// Mitsubishi GX Works2 project: pcl_6   PLC: FX3G

// global labels: Global1
VAR_GLOBAL
  start_day AT X010 : BOOL;
  finish_bread AT M1 : BOOL;
  finish_hala AT M1 : BOOL;
  flour_start_day AT D1100 : REAL;
END_VAR
VAR_GLOBAL CONSTANT
  min_flour : REAL := 100;
END_VAR
VAR_GLOBAL
  is_flour_enough AT M2 : BOOL;
  yeast AT D1200 : REAL;
  flour AT D1100 : REAL;
END_VAR
VAR_GLOBAL CONSTANT
  precent_at_least_5 : REAL := 5;
  precent_at_least_1hlcey5 : REAL := 5;
  precent_at_least_1hlcey2 : REAL := 2;
END_VAR
VAR_GLOBAL
  water AT D1300 : REAL;
END_VAR
VAR_GLOBAL CONSTANT
  hlcey5 : REAL := 5;
  hlcey2 : REAL := 2;
  caul0_3 : REAL := 0.3;
END_VAR
VAR_GLOBAL
  oil AT D1400 : REAL;
END_VAR
VAR_GLOBAL CONSTANT
  caful0_3 : REAL := 0.3;
END_VAR
VAR_GLOBAL
  spises AT D1500 : REAL;
END_VAR
VAR_GLOBAL CONSTANT
  caful0_1 : REAL := 0.1;
END_VAR
VAR_GLOBAL
  is_ingredients_enough AT M3 : BOOL;
  is_water_enough AT M3 : BOOL;
  is_oil_enough AT M4 : BOOL;
  is_spices_enough AT M5 : BOOL;
  spices AT D1500 : REAL;
  is_yeast_enough AT M6 : BOOL;
  day_work AT Y010 : BOOL;
  emergency_button AT M7 : BOOL;
  emergency_button_press AT X007 : BOOL;
  BAKAR AT M9 : BOOL;
  tc1 AT TC200 : BOOL;
END_VAR
VAR_GLOBAL CONSTANT
  cons50 : INT;
  cons500 : REAL := 500;
END_VAR
VAR_GLOBAL
  ts1 AT TS200 : BOOL;
  tc AT TC201 : BOOL;
  tc2 AT TC201 : BOOL;
  ts2 AT TS201 : BOOL;
END_VAR
VAR_GLOBAL CONSTANT
  COUNTER4 : INT;
END_VAR
VAR_GLOBAL
  firctC1 AT CC1 : BOOL;
  outC AT CS1 : BOOL;
  insert_flour AT D1102 : REAL;
  insert_yeast AT D1202 : REAL;
  insert_water AT D1302 : REAL;
  insert_oil AT D1402 : REAL;
  insert_spices AT D1502 : REAL;
  PREPARING AT X002 : BOOL;
  TimerPrep AT TC6 : BOOL;
END_VAR
VAR_GLOBAL CONSTANT
  PT3000 : REAL := 3000;
END_VAR
VAR_GLOBAL
  Lamp_Prepare AT Y005 : BOOL;
  LISHA AT M10 : BOOL;
  TIMER_OFF AT X001 : BOOL;
  NOTY AT Y005 : BOOL;
  SWITCH1 AT X001 : BOOL;
  LAMP1 AT Y001 : BOOL;
  SWITCH10 AT X010 : BOOL;
  RESET1 AT M10 : BOOL;
  SWITCH11 AT X011 : BOOL;
  RESET2 AT TC203 : BOOL;
END_VAR
VAR_GLOBAL CONSTANT
  PT300 : INT := 300;
END_VAR
VAR_GLOBAL
  stop_day AT M10 : BOOL;
  twoButton AT TC201 : BOOL;
  day_work_int AT M12 : BOOL;
  AEFG AT CS1 : BOOL;
  blink2 AT M50 : BOOL;
  blinkA AT TC1 : BOOL;
END_VAR
VAR_GLOBAL CONSTANT
  blinktimems : INT := 5;
END_VAR
VAR_GLOBAL
  blinktest2 AT TS1 : BOOL;
  blinkBASF AT TC2 : BOOL;
END_VAR
VAR_GLOBAL CONSTANT
  blinktimems4234 : INT := 5;
END_VAR
VAR_GLOBAL
  blinktest3 AT TS2 : BOOL;
  blink3QWER AT M55 : BOOL;
  COUN AT CC1 : BOOL;
END_VAR
VAR_GLOBAL CONSTANT
  ASDFS : INT := 6;
END_VAR
VAR_GLOBAL
  dONE_COUNT_6 AT M13 : BOOL;
  day_work_int_2 AT M14 : BOOL;
  day_END_BLINK AT M22 : BOOL;
  DOUBLE_CLICK AT CC3 : BOOL;
  HATPAHA AT X011 : BOOL;
END_VAR
VAR_GLOBAL CONSTANT
  COUNT2 : INT := 2;
END_VAR
VAR_GLOBAL
  blink_for_3 AT CS3 : BOOL;
  HATPAHa_end AT CS4 : BOOL;
  HELP1 AT M51 : BOOL;
  blink_DUR_3 AT TS3 : BOOL;
  NURA2 AT Y002 : BOOL;
  blink22 AT TC3 : BOOL;
  blin33 AT TC4 : BOOL;
  blinktest3TIMES AT TS4 : BOOL;
  NURA3 AT Y003 : BOOL;
END_VAR
VAR_GLOBAL CONSTANT
  SPIRA : INT := 6;
END_VAR
VAR_GLOBAL
  NURA4 AT TC8 : BOOL;
END_VAR
VAR_GLOBAL CONSTANT
  FOUR_SECOND : INT := 40;
END_VAR
VAR_GLOBAL
  FOUR_SEC AT TS8 : BOOL;
  Y4OPEN AT Y004 : BOOL;
  GELEM1 AT X002 : BOOL;
END_VAR
VAR_GLOBAL CONSTANT
  PT30 : INT := 30;
END_VAR
VAR_GLOBAL
  Lamp_5 AT Y005 : BOOL;
  start_lisha AT X001 : BOOL;
  thilat_hatpaha AT CS3 : BOOL;
END_VAR
VAR_GLOBAL CONSTANT
  minus100 : REAL := 100;
  minus20 : REAL := 20;
  minus50 : REAL := 50;
  minus30 : REAL := 30;
  minus10 : REAL := 10;
END_VAR
VAR_GLOBAL
  UNTIL_LISHA_DONE AT Y001 : BOOL;
  THREE_SEC_LIGHT AT TS6 : BOOL;
  LIGHT_5Y AT Y005 : BOOL;
END_VAR
VAR_GLOBAL CONSTANT
  VALUE_1 : INT := 1;
END_VAR
VAR_GLOBAL
  MIXER AT D1700 : INT;
END_VAR
VAR_GLOBAL CONSTANT
  VALUE_0 : INT;
END_VAR
VAR_GLOBAL
  hatpaha_container AT D1701 : INT;
  backing_form AT D1702 : INT;
  QUALITY_TEST AT X003 : BOOL;
  ANALOG_INPUT_2 AT D8281 : WORD;
END_VAR
VAR_GLOBAL CONSTANT
  Bigger_than_one : DINT := 400;
  Smaller_Than_Five : DINT := 2000;
END_VAR
VAR_GLOBAL
  Is_Bigger_Than_One AT M60 : BOOL;
  Is_Smaller_Than_Five AT M61 : BOOL;
  erech_analog AT D1670 : DINT;
  NURA6 AT TC9 : BOOL;
END_VAR
VAR_GLOBAL CONSTANT
  FIVE_SECONDS : INT := 50;
END_VAR
VAR_GLOBAL
  LIGHT_5_SEC AT TS9 : BOOL;
  NURA_6 AT Y006 : BOOL;
  BREAD_STRUCTURE AT D1600 : INT;
END_VAR
VAR_GLOBAL CONSTANT
  PLUS_1 : INT := 1;
END_VAR
VAR_GLOBAL
  bakery_shelves AT D1703 : INT;
  chack_twice AT CC7 : BOOL;
END_VAR
VAR_GLOBAL CONSTANT
  SPIRA_2 : INT := 2;
  Bigger_than_five : DINT := 2000;
  Smaller_Than_one : DINT := 400;
END_VAR
VAR_GLOBAL
  Is_Bigger_Than_five AT M60 : BOOL;
  Is_Smaller_Than_one AT M61 : BOOL;
  TIful AT M63 : BOOL;
  hathel AT M63 : BOOL;
END_VAR
VAR_GLOBAL CONSTANT
  zero : DINT;
END_VAR
VAR_GLOBAL
  hivhuv_end AT CC4 : BOOL;
  chacked_twice AT CS7 : BOOL;
  Bitahon AT M67 : BOOL;
END_VAR
VAR_GLOBAL CONSTANT
  VALUE_0_DW : DINT;
  VALUE_0_bit : BOOL;
END_VAR

// task Task_01 (event TRUE, interval 0, priority 31): POU_01

PROGRAM POU_01
(* structured ladder/FBD written out as ST: instructions are called as NAME(EN, inputs, outputs); _pN, _eN, _tN stand for wires *)
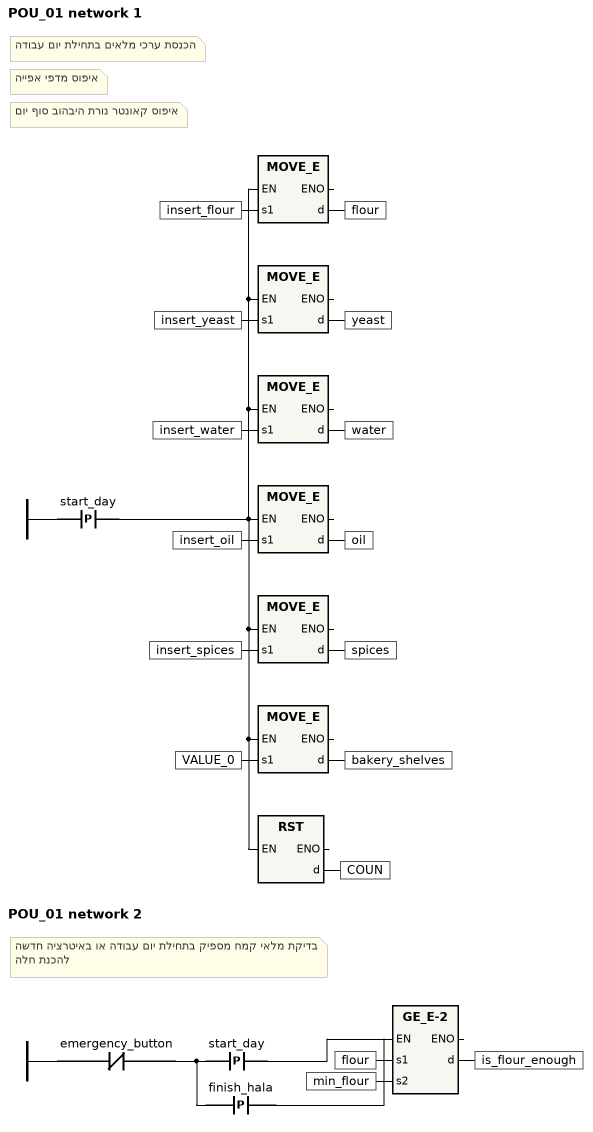
(* network 1 *)
(* הכנסת ערכי מלאים בתחילת יום עבודה *)
(* איפוס מדפי אפייה *)
(* איפוס קאונטר נורת היבהוב סוף יום *)
_p1 := LDP(TRUE, start_day);
MOVE_E(_p1, insert_flour, flour);
MOVE_E(_p1, insert_yeast, yeast);
MOVE_E(_p1, insert_water, water);
MOVE_E(_p1, insert_oil, oil);
MOVE_E(_p1, insert_spices, spices);
MOVE_E(_p1, VALUE_0, bakery_shelves);
RST(_p1, COUN);
(* network 2 *)
(* בדיקת מלאי קמח מספיק בתחילת יום עבודה או באיטרציה חדשה להכנת חלה *)
_p1 := NOT emergency_button;
GE_E((_p1 AND LDP(TRUE, start_day)) OR (_p1 AND LDP(TRUE, finish_hala)), flour, min_flour, is_flour_enough);
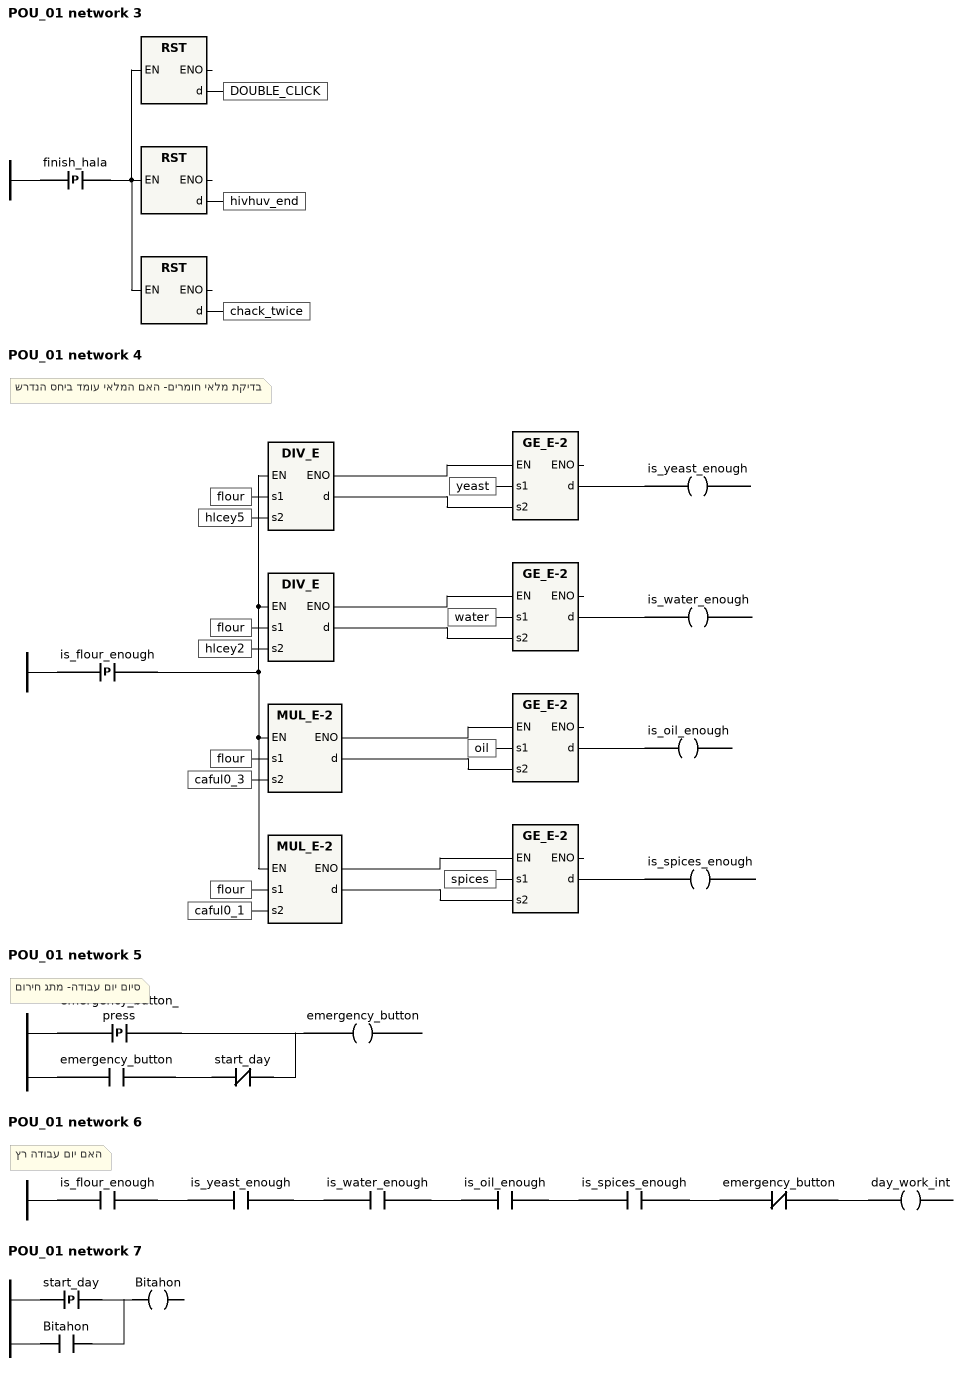
(* network 3 *)
_p1 := LDP(TRUE, finish_hala);
RST(_p1, DOUBLE_CLICK);
RST(_p1, hivhuv_end);
RST(_p1, chack_twice);
(* network 4 *)
(* בדיקת מלאי חומרים- האם המלאי עומד ביחס הנדרש *)
_p1 := LDP(TRUE, is_flour_enough);
_e3 := DIV_E(_p1, flour, hlcey5, _t2);
GE_E(_e3, yeast, _t2, _t4);
is_yeast_enough := _t4;
_e6 := DIV_E(_p1, flour, hlcey2, _t5);
GE_E(_e6, water, _t5, _t7);
is_water_enough := _t7;
_e9 := MUL_E(_p1, flour, caful0_3, _t8);
GE_E(_e9, oil, _t8, _t10);
is_oil_enough := _t10;
_e12 := MUL_E(_p1, flour, caful0_1, _t11);
GE_E(_e12, spices, _t11, _t13);
is_spices_enough := _t13;
(* network 5 *)
(* סיום יום עבודה- מתג חירום *)
emergency_button := LDP(TRUE, emergency_button_press) OR (emergency_button AND NOT start_day);
(* network 6 *)
(* האם יום עבודה רץ *)
day_work_int := is_flour_enough AND is_yeast_enough AND is_water_enough AND is_oil_enough AND is_spices_enough AND NOT emergency_button;
(* network 7 *)
Bitahon := LDP(TRUE, start_day) OR Bitahon;
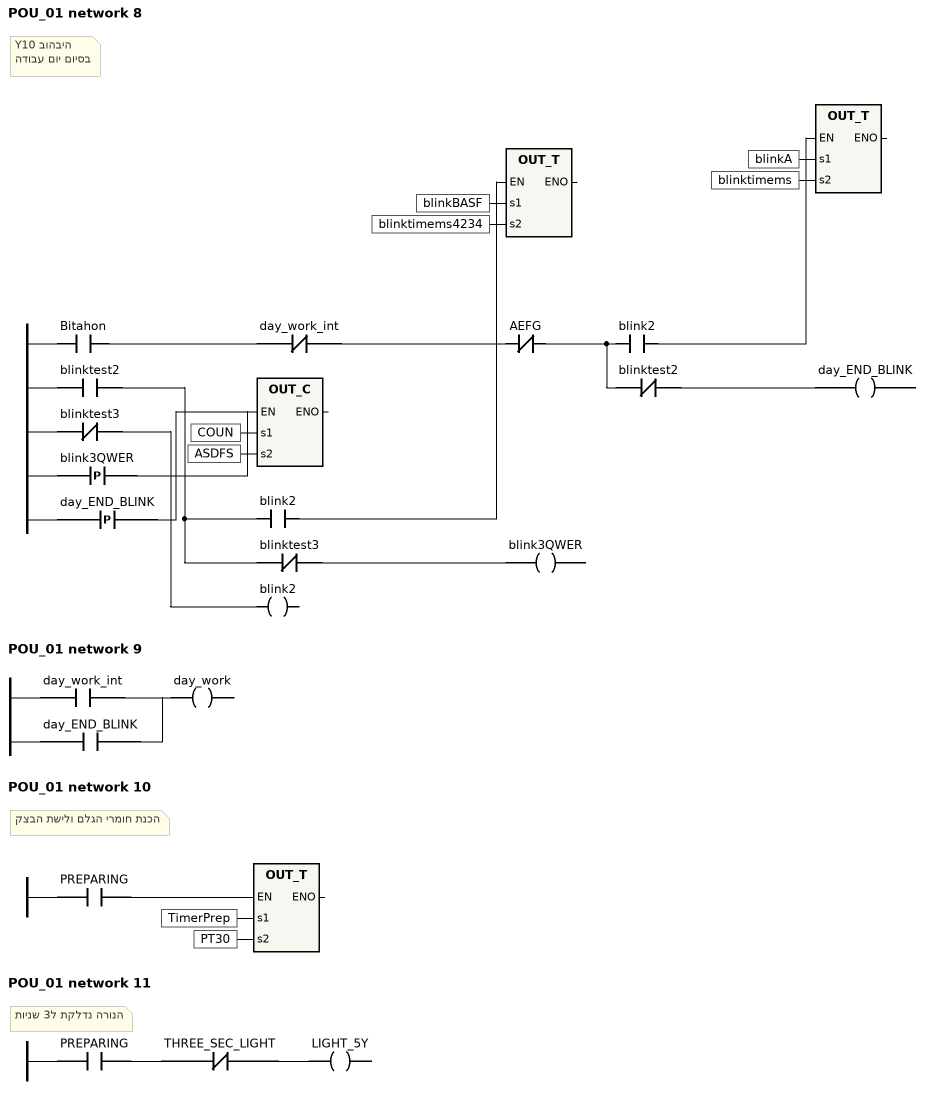
(* network 8 *)
(* היבהוב Y10 /  בסיום יום עבודה *)
_p1 := Bitahon AND NOT day_work_int AND NOT AEFG;
OUT_T(_p1 AND blink2, blinkA, blinktimems);
day_END_BLINK := _p1 AND NOT blinktest2;
OUT_T(blinktest2 AND blink2, blinkBASF, blinktimems4234);
blink3QWER := blinktest2 AND NOT blinktest3;
blink2 := NOT blinktest3;
OUT_C(LDP(TRUE, blink3QWER) OR LDP(TRUE, day_END_BLINK), COUN, ASDFS);
(* network 9 *)
day_work := day_work_int OR day_END_BLINK;
(* network 10 *)
(* הכנת חומרי הגלם ולישת הבצק *)
OUT_T(PREPARING, TimerPrep, PT30);
(* network 11 *)
(* הנורה נדלקת ל3 שניות *)
LIGHT_5Y := PREPARING AND NOT THREE_SEC_LIGHT;
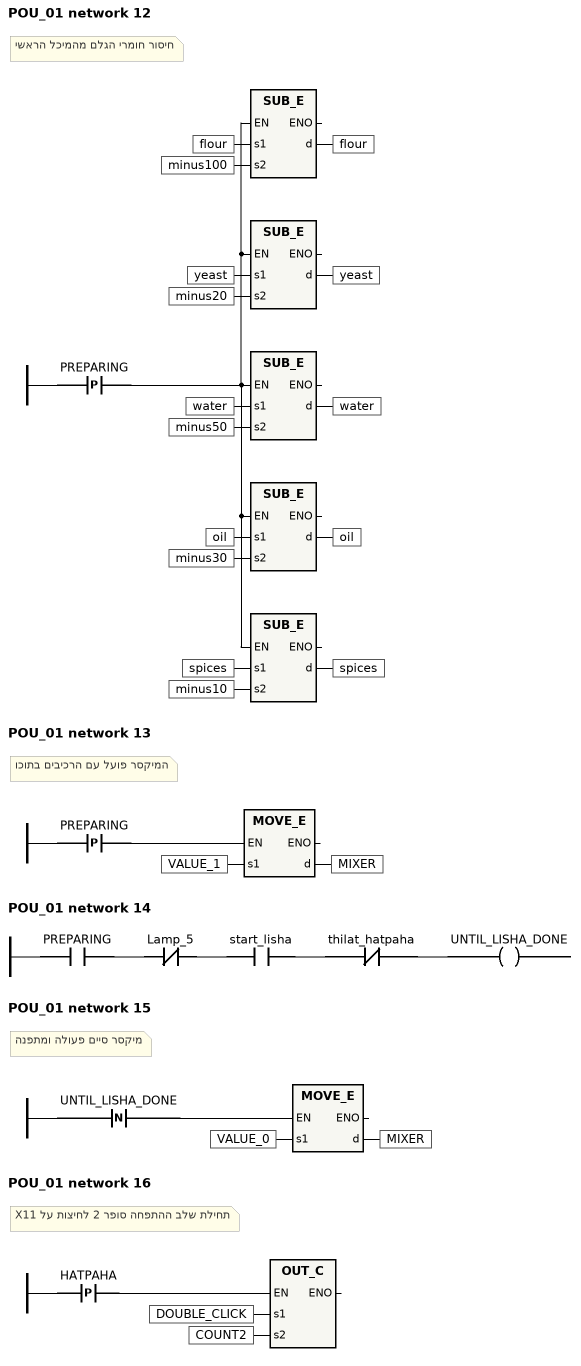
(* network 12 *)
(* חיסור חומרי הגלם מהמיכל הראשי *)
_p1 := LDP(TRUE, PREPARING);
SUB_E(_p1, flour, minus100, flour);
SUB_E(_p1, yeast, minus20, yeast);
SUB_E(_p1, water, minus50, water);
SUB_E(_p1, oil, minus30, oil);
SUB_E(_p1, spices, minus10, spices);
(* network 13 *)
(* המיקסר פועל עם הרכיבים בתוכו *)
MOVE_E(LDP(TRUE, PREPARING), VALUE_1, MIXER);
(* network 14 *)
UNTIL_LISHA_DONE := PREPARING AND NOT Lamp_5 AND start_lisha AND NOT thilat_hatpaha;
(* network 15 *)
(* מיקסר סיים פעולה ומתפנה *)
MOVE_E(LDF(TRUE, UNTIL_LISHA_DONE), VALUE_0, MIXER);
(* network 16 *)
(* תחילת שלב ההתפחה סופר 2 לחיצות על X11 *)
OUT_C(LDP(TRUE, HATPAHA), DOUBLE_CLICK, COUNT2);
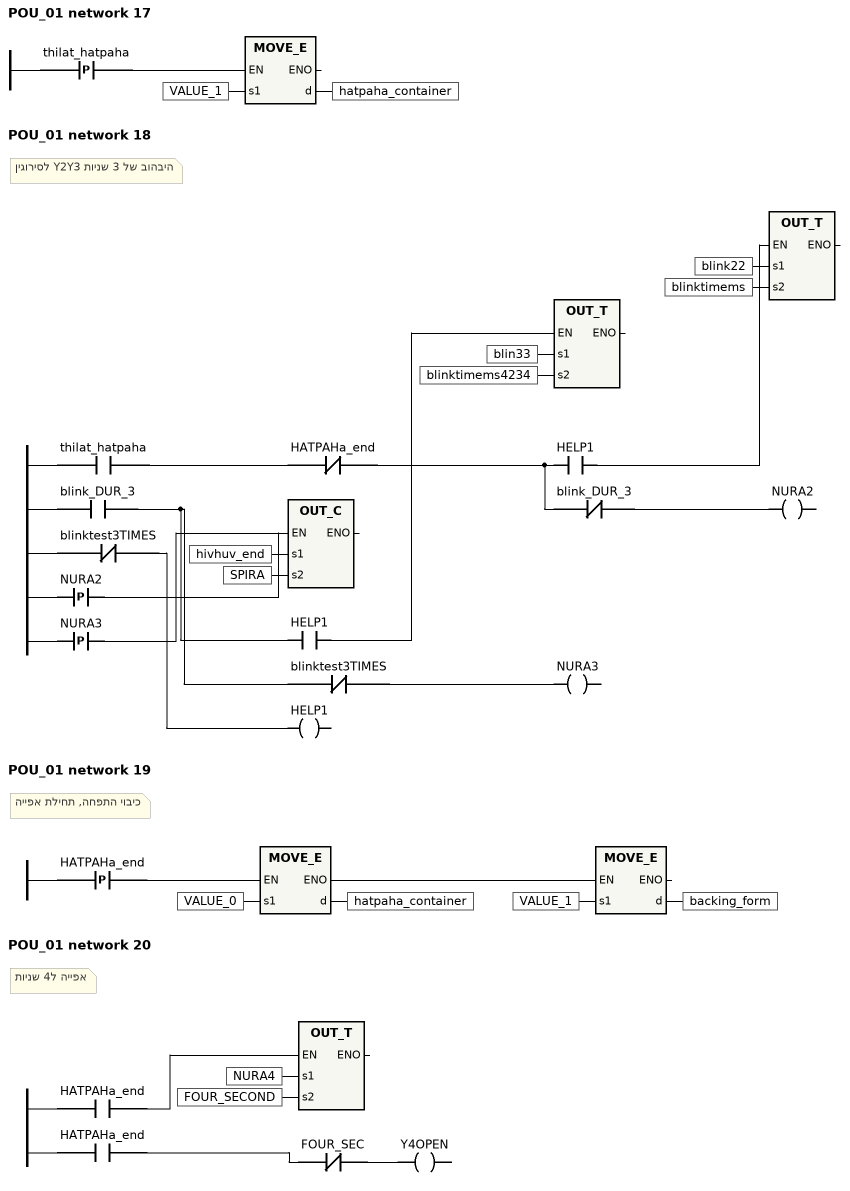
(* network 17 *)
MOVE_E(LDP(TRUE, thilat_hatpaha), VALUE_1, hatpaha_container);
(* network 18 *)
(* היבהוב של 3 שניות Y2Y3 לסירוגין *)
_p1 := thilat_hatpaha AND NOT HATPAHa_end;
OUT_T(_p1 AND HELP1, blink22, blinktimems);
NURA2 := _p1 AND NOT blink_DUR_3;
OUT_T(blink_DUR_3 AND HELP1, blin33, blinktimems4234);
NURA3 := blink_DUR_3 AND NOT blinktest3TIMES;
HELP1 := NOT blinktest3TIMES;
OUT_C(LDP(TRUE, NURA2) OR LDP(TRUE, NURA3), hivhuv_end, SPIRA);
(* network 19 *)
(* כיבוי התפחה, תחילת אפייה *)
_e1 := MOVE_E(LDP(TRUE, HATPAHa_end), VALUE_0, hatpaha_container);
MOVE_E(_e1, VALUE_1, backing_form);
(* network 20 *)
(* אפייה ל4 שניות *)
OUT_T(HATPAHa_end, NURA4, FOUR_SECOND);
Y4OPEN := HATPAHa_end AND NOT FOUR_SEC;
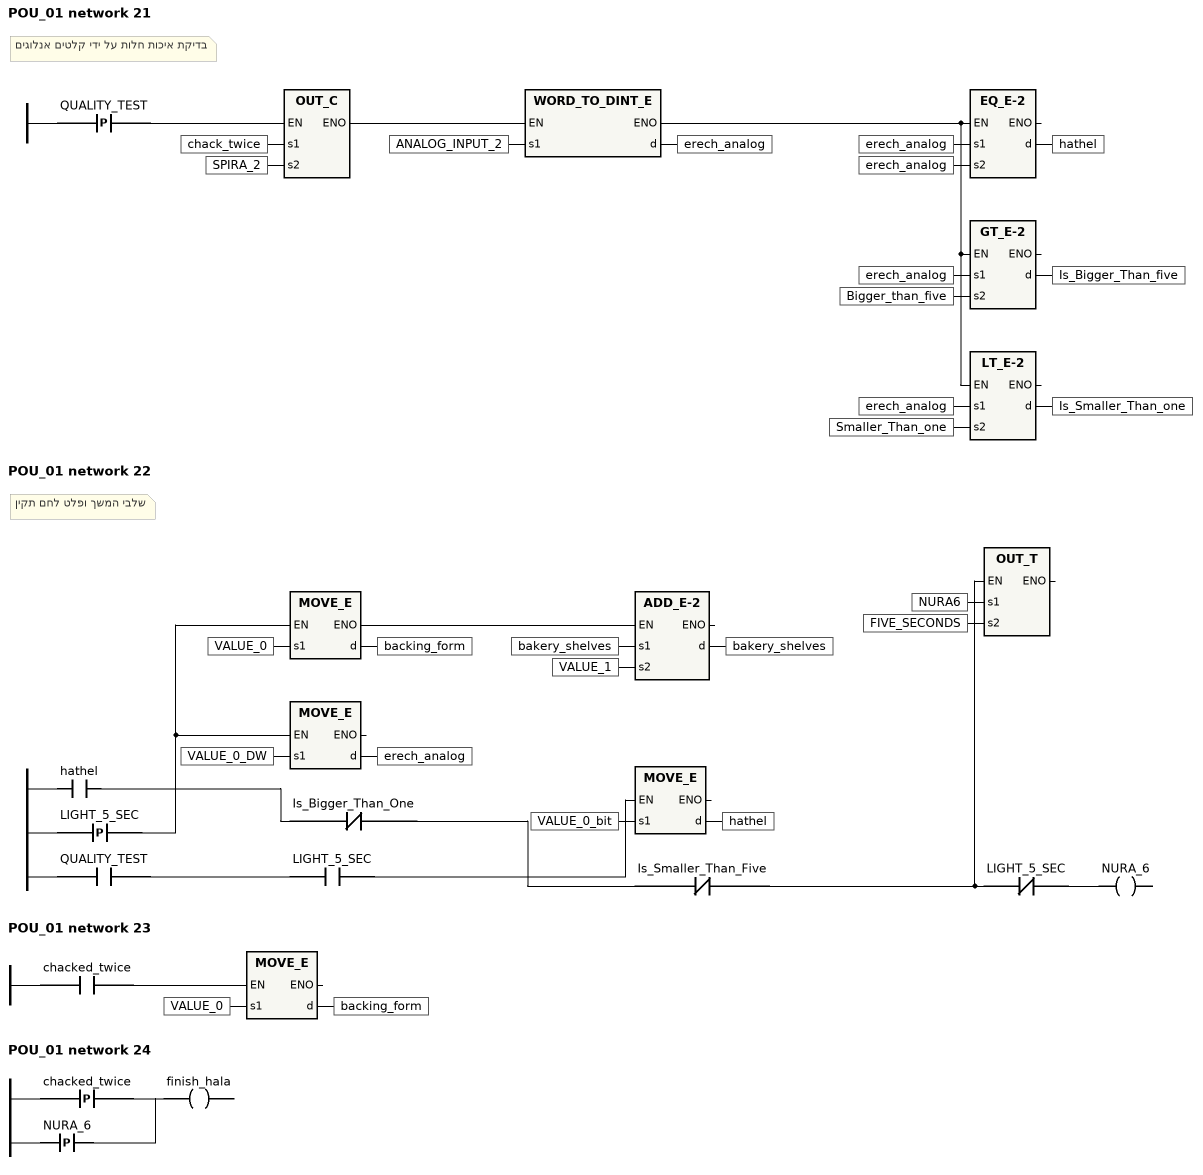
(* network 21 *)
(* בדיקת איכות חלות על ידי קלטים אנלוגים *)
_e1 := OUT_C(LDP(TRUE, QUALITY_TEST), chack_twice, SPIRA_2);
_e2 := WORD_TO_DINT_E(_e1, ANALOG_INPUT_2, erech_analog);
EQ_E(_e2, erech_analog, erech_analog, hathel);
GT_E(_e2, erech_analog, Bigger_than_five, Is_Bigger_Than_five);
LT_E(_e2, erech_analog, Smaller_Than_one, Is_Smaller_Than_one);
(* network 22 *)
(* שלבי המשך ופלט לחם תקין *)
_p1 := hathel AND NOT Is_Bigger_Than_One AND NOT Is_Smaller_Than_Five;
OUT_T(_p1, NURA6, FIVE_SECONDS);
NURA_6 := _p1 AND NOT LIGHT_5_SEC;
_p2 := LDP(TRUE, LIGHT_5_SEC);
_e3 := MOVE_E(_p2, VALUE_0, backing_form);
ADD_E(_e3, bakery_shelves, VALUE_1, bakery_shelves);
MOVE_E(_p2, VALUE_0_DW, erech_analog);
MOVE_E(QUALITY_TEST AND LIGHT_5_SEC, VALUE_0_bit, hathel);
(* network 23 *)
MOVE_E(chacked_twice, VALUE_0, backing_form);
(* network 24 *)
finish_hala := LDP(TRUE, chacked_twice) OR LDP(TRUE, NURA_6);
END_PROGRAM
